TYPE ST_AXIS_TORQUE :
STRUCT
END_STRUCT
END_TYPE

(* stored: Version 1.1.0.1, ProductVersion 3.1.4024.11
   DUT ST_AXIS_TORQUE: Id {f16439d9-9fc6-4a22-8068-f69f84308fe5} *)
